(* PLC project LibIT_EEPROM, lamsystems-it.ru LibIT_EEPROM 1 *)
(* stored: creationDateTime 2019-11-13T09:37:45, productRelease 0, modificationDateTime 2021-12-10T18:05:31, version 1 *)

TYPE EeRegByte : STRUCT
  Addr : DINT := -1;
  Ty : BYTE := 1;
END_STRUCT;
END_TYPE

TYPE EeRegWord : STRUCT
  Addr : DINT := -1;
  Ty : BYTE := 2;
END_STRUCT;
END_TYPE

TYPE EeRegDWord : STRUCT
  Addr : DINT := -1;
  Ty : BYTE := 3;
END_STRUCT;
END_TYPE

TYPE EeRegLWord : STRUCT
  Addr : DINT := -1;
  Ty : BYTE := 4;
END_STRUCT;
END_TYPE

TYPE EeRegReal : STRUCT
  Addr : DINT := -1;
  Ty : BYTE := 5;
END_STRUCT;
END_TYPE

TYPE EeRegLReal : STRUCT
  Addr : DINT := -1;
  Ty : BYTE := 6;
END_STRUCT;
END_TYPE

FUNCTION_BLOCK EeReadLReal
  VAR_INPUT
    Ex : BOOL := FALSE;
    Reg : EeRegLReal;
  END_VAR
  VAR_OUTPUT
    OVal : LREAL := 0.0;
    Ok : BYTE := 0;
  END_VAR

            {extern void AppEe_Read(EEREADLREAL*);AppEe_Read(data__);}

          
END_FUNCTION_BLOCK

FUNCTION_BLOCK EeReadByte
  VAR_INPUT
    Ex : BOOL := FALSE;
    Reg : EeRegByte;
  END_VAR
  VAR_OUTPUT
    OVal : BYTE := 0;
    Ok : BYTE := 0;
  END_VAR
  VAR
    RegLReal : EeRegLReal;
    Func : EeReadLReal;
  END_VAR

            RegLReal.Addr:= Reg.Addr;
RegLReal.Ty:= Reg.Ty;
Func(Ex:=Ex, Reg:=RegLReal);
OVal:= LREAL_TO_BYTE(Func.OVal);
Ok:= Func.Ok;
          
END_FUNCTION_BLOCK

FUNCTION_BLOCK EeReadWord
  VAR_INPUT
    Ex : BOOL := FALSE;
    Reg : EeRegWord;
  END_VAR
  VAR_OUTPUT
    OVal : WORD := 0;
    Ok : BYTE := 0;
  END_VAR
  VAR
    RegLReal : EeRegLReal;
    Func : EeReadLReal;
  END_VAR

            RegLReal.Addr:= Reg.Addr;
RegLReal.Ty:= Reg.Ty;
Func(Ex:=Ex, Reg:=RegLReal);
OVal:= LREAL_TO_WORD(Func.OVal);
Ok:= Func.Ok;
          
END_FUNCTION_BLOCK

FUNCTION_BLOCK EeReadDWord
  VAR_INPUT
    Ex : BOOL := FALSE;
    Reg : EeRegDWord;
  END_VAR
  VAR_OUTPUT
    OVal : DWORD := 0;
    Ok : BYTE := 0;
  END_VAR
  VAR
    RegLReal : EeRegLReal;
    Func : EeReadLReal;
  END_VAR

            RegLReal.Addr:= Reg.Addr;
RegLReal.Ty:= Reg.Ty;
Func(Ex:=Ex, Reg:=RegLReal);
OVal:= LREAL_TO_DWORD(Func.OVal);
Ok:= Func.Ok;
          
END_FUNCTION_BLOCK

FUNCTION_BLOCK EeReadLWord
  VAR_INPUT
    Ex : BOOL := FALSE;
    Reg : EeRegLWord;
  END_VAR
  VAR_OUTPUT
    OVal : LWORD := 0;
    Ok : BYTE := 0;
  END_VAR
  VAR
    RegLReal : EeRegLReal;
    Func : EeReadLReal;
  END_VAR

            RegLReal.Addr:= Reg.Addr;
RegLReal.Ty:= Reg.Ty;
Func(Ex:=Ex, Reg:=RegLReal);
OVal:= LREAL_TO_LWORD(Func.OVal);
Ok:= Func.Ok;
          
END_FUNCTION_BLOCK

FUNCTION_BLOCK EeReadReal
  VAR_INPUT
    Ex : BOOL := FALSE;
    Reg : EeRegReal;
  END_VAR
  VAR_OUTPUT
    OVal : REAL := 0.0;
    Ok : BYTE := 0;
  END_VAR
  VAR
    RegLReal : EeRegLReal;
    Func : EeReadLReal;
  END_VAR

            RegLReal.Addr:= Reg.Addr;
RegLReal.Ty:= Reg.Ty;
Func(Ex:=Ex, Reg:=RegLReal);
OVal:= LREAL_TO_REAL(Func.OVal);
Ok:= Func.Ok;
          
END_FUNCTION_BLOCK

FUNCTION_BLOCK EeWriteLReal
  VAR_INPUT
    Ex : BOOL := FALSE;
    Reg : EeRegLReal;
    Val : LREAL := 0.0;
  END_VAR
  VAR_OUTPUT
    Ok : BYTE := 0;
  END_VAR

            {extern void AppEe_Write(EEWRITELREAL*);AppEe_Write(data__);}
          
END_FUNCTION_BLOCK

FUNCTION_BLOCK EeWriteByte
  VAR_INPUT
    Ex : BOOL := FALSE;
    Reg : EeRegByte;
    Val : BYTE := 0;
  END_VAR
  VAR_OUTPUT
    Ok : BYTE := 0;
  END_VAR
  VAR
    RegLReal : EeRegLReal;
    Func : EeWriteLReal;
  END_VAR

            RegLReal.Addr:= Reg.Addr;
RegLReal.Ty:= Reg.Ty;
Func(Ex:=Ex, Reg:=RegLReal, Val:=BYTE_TO_LREAL(Val));
Ok:= Func.Ok;
          
END_FUNCTION_BLOCK

FUNCTION_BLOCK EeWriteWord
  VAR_INPUT
    Ex : BOOL := FALSE;
    Reg : EeRegWord;
    Val : WORD := 0;
  END_VAR
  VAR_OUTPUT
    Ok : BYTE := 0;
  END_VAR
  VAR
    RegLReal : EeRegLReal;
    Func : EeWriteLReal;
  END_VAR

            RegLReal.Addr:= Reg.Addr;
RegLReal.Ty:= Reg.Ty;
Func(Ex:=Ex, Reg:=RegLReal, Val:=WORD_TO_LREAL(Val));
Ok:= Func.Ok;
          
END_FUNCTION_BLOCK

FUNCTION_BLOCK EeWriteDWord
  VAR_INPUT
    Ex : BOOL := FALSE;
    Reg : EeRegDWord;
    Val : DWORD := 0;
  END_VAR
  VAR_OUTPUT
    Ok : BYTE := 0;
  END_VAR
  VAR
    RegLReal : EeRegLReal;
    Func : EeWriteLReal;
  END_VAR

            RegLReal.Addr:= Reg.Addr;
RegLReal.Ty:= Reg.Ty;
Func(Ex:=Ex, Reg:=RegLReal, Val:=DWORD_TO_LREAL(Val));
Ok:= Func.Ok;
          
END_FUNCTION_BLOCK

FUNCTION_BLOCK EeWriteLWord
  VAR_INPUT
    Ex : BOOL := FALSE;
    Reg : EeRegLWord;
    Val : LWORD := 0;
  END_VAR
  VAR_OUTPUT
    Ok : BYTE := 0;
  END_VAR
  VAR
    RegLReal : EeRegLReal;
    Func : EeWriteLReal;
  END_VAR

            RegLReal.Addr:= Reg.Addr;
RegLReal.Ty:= Reg.Ty;
Func(Ex:=Ex, Reg:=RegLReal, Val:=LWORD_TO_LREAL(Val));
Ok:= Func.Ok;
          
END_FUNCTION_BLOCK

FUNCTION_BLOCK EeWriteReal
  VAR_INPUT
    Ex : BOOL := FALSE;
    Reg : EeRegReal;
    Val : REAL := 0.0;
  END_VAR
  VAR_OUTPUT
    Ok : BYTE := 0;
  END_VAR
  VAR
    RegLReal : EeRegLReal;
    Func : EeWriteLReal;
  END_VAR

            RegLReal.Addr:= Reg.Addr;
RegLReal.Ty:= Reg.Ty;
Func(Ex:=Ex, Reg:=RegLReal, Val:=REAL_TO_LREAL(Val));
Ok:= Func.Ok;
          
END_FUNCTION_BLOCK
